{attribute 'linkalways'} 
{attribute 'no_explicit_call' := 'This FB is a CLASS and must be accessed using methods or properties'}
{attribute 'enable_dynamic_creation'}
FUNCTION_BLOCK _Array0to1OfSINT EXTENDS ArrayDatatypeBase_1D
VAR CONSTANT
	lBound : DINT := 0;
	uBound : DINT := 1;
END_VAR
VAR
	localData : ARRAY [lBound..uBound] OF SINT;
	activeData : REFERENCE TO ARRAY [lBound..uBound] OF SINT REF= localData;
	elements : ARRAY [lBound..uBound] OF _SINT(0);
	baseType : _SINT(0);
END_VAR

PROPERTY PUBLIC Address : PVOID
GET
Address := ADR(activeData);
END_GET
END_PROPERTY

PROPERTY PUBLIC BaseDatatype : I_Datatype
GET
BaseDatatype := baseType;
END_GET
END_PROPERTY

METHOD PUBLIC ClearReference
VAR_INPUT
END_VAR
activeData REF= localData;
SetElementReference();
END_METHOD

METHOD PUBLIC Clone : I_Datatype
VAR
    pClone : POINTER TO _Array0to1OfSINT;
END_VAR
pClone := __NEW(_Array0to1OfSINT());
pClone^.Value := Value;
Clone := pClone^;
END_METHOD

METHOD FB_init : BOOL
VAR_INPUT
	bInitRetains : BOOL; // if TRUE, the retain variables are initialized (warm start / cold start)
	bInCopyCode : BOOL;  // if TRUE, the instance afterwards gets moved into the copy code (online change)
END_VAR
SetElementReference();
END_METHOD

METHOD PUBLIC MakeReferenceTo
VAR_INPUT
	ReferenceTarget : REFERENCE TO ARRAY [lBound..uBound] OF SINT;
END_VAR
activeData REF= ReferenceTarget;
SetElementReference();
END_METHOD

METHOD PROTECTED OnSerializeArrayValues
VAR_INPUT
	Serializer : I_Serializer;
END_VAR
VAR
	i : DINT;
END_VAR
FOR i := lBound TO uBound DO
	elements[i].SerializeWith(Serializer);
END_FOR
END_METHOD

METHOD PROTECTED SetElementReference
VAR_INPUT
END_VAR
VAR
	i : DINT;
END_VAR
FOR i := lBound TO uBound DO
	elements[i].MakeReferenceTo(activeData[i]);
END_FOR
END_METHOD

PROPERTY PUBLIC Size : UDINT
GET
Size := SIZEOF(activeData);
END_GET
END_PROPERTY

METHOD PROTECTED TryDeserializeArrayValues : BOOL
VAR_INPUT
	Deserializer : I_Deserializer;
	Feedback : I_DeserializerFeedback;
END_VAR
VAR
	enumerator : I_DeserializerArrayForwardEnumerator;
	i : DINT;
END_VAR
enumerator := Deserializer.GetArrayEnumerator();
i := lBound;

WHILE enumerator.MoveNext() AND i <= uBound DO
	
	IF NOT elements[i].TryDeserializeFrom(enumerator.Current, Feedback) THEN
		EXIT;
	END_IF
	i := i + 1;

END_WHILE
enumerator.Dispose();
END_METHOD

METHOD PUBLIC TryGetElementAsDatatypeByIndex : BOOL
VAR_INPUT
	Index : DINT;
	Destination : REFERENCE TO I_Datatype;
END_VAR
IF Index < lbound OR Index > ubound THEN
	RETURN;
END_IF

Destination := elements[Index];
TryGetElementAsDatatypeByIndex := TRUE;
END_METHOD

METHOD PUBLIC TryGetLowerBound : BOOL
VAR_INPUT
	Dimention : UDINT;
	Destination : REFERENCE TO DINT;
END_VAR
IF Dimention = 1 THEN
	Destination := lBound;
	TryGetLowerBound := TRUE;
END_IF
END_METHOD

METHOD PUBLIC TryGetUpperBound : BOOL
VAR_INPUT
	Dimention : UDINT;
	Destination : REFERENCE TO DINT;
END_VAR
IF Dimention = 1 THEN
	Destination := uBound;
	TryGetUpperBound := TRUE;
END_IF
END_METHOD

METHOD TryMakeReferenceTo : BOOL
VAR_INPUT
	Target : I_Datatype;
END_VAR
VAR
	targetAsArray : I_ArrayDatatype;
	pTargetData : POINTER TO ARRAY [lBound..uBound] OF SINT;
END_VAR
IF NOT Target.TryResolveAsArrayDatatype(targetAsArray) THEN
	RETURN;
END_IF

IF NOT (targetAsArray.Identifier = Identifier) THEN
	RETURN;
END_IF

pTargetData := Target.Address;
activeData REF= pTargetData^;
SetElementReference();
TryMakeReferenceTo := TRUE;
END_METHOD

PROPERTY PUBLIC Value : REFERENCE TO ARRAY [lBound..uBound] OF SINT;
GET
Value ref= activeData;
END_GET
END_PROPERTY

END_FUNCTION_BLOCK

(* stored: Version 1.1.0.1, ProductVersion 3.1.4024.13
   POU _Array0to1OfSINT: Id {b74b1364-df5e-0828-0a46-1ade6ed70ae4}, SpecialFunc None
   Folder Core: Id {90f0a20f-d4e5-053a-3302-f78d05041d03}
   Folder Constructor: Id {af112035-4d02-0fe4-3318-30b59465df02}
   Folder Protected: Id {62a519e0-f767-06c3-174c-2ac944836ec3}
   Folder Customize: Id {a9fce513-07f2-0f01-25a4-d6f9e02303ab}
   Property Address: Id {2262a991-f639-0acf-32ed-ee85af652aa5}
   Get Get: Id {dc1babc3-12f3-02b9-1bd2-2460292c5565}
   Property BaseDatatype: Id {6dbe1356-79b1-0411-3fe9-8cb1e5e0532c}
   Get Get: Id {877ab87a-82cf-0d12-119d-efee93d93cee}
   Method ClearReference: Id {911cb6bb-3291-02ff-32d2-461466730fbb}
   Method Clone: Id {538e6725-9a2f-0d23-164f-1919bf8783b1}
   Method FB_init: Id {80262695-a2c8-01f1-34d5-564b6b189834}
   Method MakeReferenceTo: Id {b14b06a0-d2c7-06b3-2c05-9f9e3496d2b4}
   Method OnSerializeArrayValues: Id {d1f6c845-4688-09a2-379a-80635823ae46}
   Method SetElementReference: Id {90803714-670c-00ba-1d15-3243993166bf}
   Property Size: Id {3b41f56b-b04d-07a0-3087-60cbd4dbb104}
   Get Get: Id {14f53b79-8cc0-0548-2581-cd32c3e5e7c0}
   Method TryDeserializeArrayValues: Id {3f3c8932-9d81-0dac-2c88-a557892ce6a7}
   Method TryGetElementAsDatatypeByIndex: Id {3a314029-56b1-044f-307b-43fc53ccafd4}
   Method TryGetLowerBound: Id {ffe8c5b3-81a4-082c-1ef3-56568208e52b}
   Method TryGetUpperBound: Id {002e3943-e767-0130-2b1c-1eb1e172315c}
   Method TryMakeReferenceTo: Id {9e2ff2db-7736-0297-202e-b7fbb89a7be2}
   Property Value: Id {8e1bed30-3c2b-07b5-22f8-9e21bdbd0de6}
   Get Get: Id {a332e3ca-081d-07f1-12cf-aefb6722d3af} *)
